INTERFACE I_MasterArmCtrl

PROPERTY isFinished : bool
GET
END_GET
END_PROPERTY

METHOD reset : BOOL
VAR_INPUT
END_VAR
END_METHOD

METHOD run : BOOL
VAR_INPUT
	monitorAngle :LREAL;
	slaveIdx :INT;
END_VAR

VAR_IN_OUT CONSTANT
	i_masterArm :FB_MasterArm;
	i_slaveStatus :ST_SlaveStatus;
END_VAR
VAR_IN_OUT
	r_masterArmCtrlCmd :ST_ArmCtrlCmds;
END_VAR
END_METHOD

END_INTERFACE

(* stored: Version 1.1.0.1, ProductVersion 3.1.4024.12
   Itf I_MasterArmCtrl: Id {f0c76191-353c-4edd-a51a-aab3c6b7f25c}
   Property isFinished: Id {4248d833-c6dc-4e42-9d08-141fd83355a1}
   Get Get: Id {7e481075-d3b2-4bb7-a7b6-ff6c734930d2}
   Method reset: Id {d3d01b04-dfab-450f-8fd4-a152b95c8241}
   Method run: Id {cdc1ac69-5bc1-4174-b158-da097af4b3d6} *)
